INTERFACE ITF_Veiligheidsmat

PROPERTY Actief : BOOL
GET
END_GET
END_PROPERTY

PROPERTY Error : BOOL
GET
END_GET
END_PROPERTY

PROPERTY Status : E_VeiligheidsmatStatus
GET
END_GET
END_PROPERTY

METHOD Update : BOOL
VAR_INPUT
END_VAR
END_METHOD

END_INTERFACE

(* stored: Version 1.1.0.1
   Itf ITF_Veiligheidsmat: Id {038ec8f4-7771-45da-90b9-22cac9b667d8}
   Property Actief: Id {45ac85ea-6f41-4dfa-9d76-998fae6ece0c}
   Get Get: Id {56f0d4cf-4573-4ccc-9600-691bb92ce950}
   Property Error: Id {7413dc96-b84c-41b2-b8c4-c7cc08e81cd2}
   Get Get: Id {97c8fbcc-6e97-4497-9321-1115c3700285}
   Property Status: Id {0557f6a8-d735-4fae-8981-51450c28851a}
   Get Get: Id {efeba6c4-1ced-409c-82a1-4b6cc78121b0}
   Method Update: Id {e0fe07c2-c9d7-412d-b19d-9a79ab3c3b70} *)
